PROGRAM MAIN
VAR
END_VAR

END_PROGRAM

(* stored: Version 1.1.0.1
   POU MAIN: Id {7b4518f5-626f-453e-8ddd-cc47dee66309} *)
